{attribute 'qualified_only'}
{attribute 'strict'}
TYPE ST_LaudaPendingCommand :
STRUCT
	Command		: Tc2_System.T_MaxString;	// Command to be send
	Value		: REAL ;	// If command has parameters, set them here. Conversion is done internally
END_STRUCT
END_TYPE

(* stored: Version 1.1.0.1, ProductVersion 3.1.4024.13
   DUT ST_LaudaPendingCommand: Id {76f478e6-3281-437b-8fdc-ae63251578dd} *)
